FUNCTION_BLOCK FB_SaMElementComplete EXTENDS FB_SaMElement
VAR
END_VAR

METHOD FB_init : BOOL
VAR_INPUT
	bInitRetains : BOOL; // if TRUE, the retain variables are initialized (warm start / cold start)
	bInCopyCode : BOOL;  // if TRUE, the instance afterwards gets moved into the copy code (online change)
END_VAR
THIS^.SetText (eLocation := E_BaseLocation.pl, wsDescription := "Kompletny");
THIS^.SetText (eLocation := E_BaseLocation.en, wsDescription := "Complete");
THIS^.SetText (eLocation := E_BaseLocation.de, wsDescription := "Vollständig");
THIS^.SetName (stName := THIS^.GetTexts ());
END_METHOD

METHOD PUBLIC InvokeStateForTopElement : BOOL
VAR_INPUT
	itfTopElement		: ITF_BaseSaMStateMethod;
END_VAR
InvokeStateForTopElement	:= itfTopElement.SP_Complete ();
END_METHOD

END_FUNCTION_BLOCK

(* stored: Version 1.1.0.1
   POU FB_SaMElementComplete: Id {49eede30-1d45-0fd6-0104-d3de73573ec2}, SpecialFunc None
   Method FB_init: Id {396c4f3a-dac3-05e5-3c6a-6c3d8bd3e42d}
   Method InvokeStateForTopElement: Id {72e8f316-2302-01df-2051-93c2d20c009a} *)
